Staubli VAL3: _incrementCol.pgx

program _incrementCol(string& x_sColValue[], bool& x_bError[])
  local num l_nColAsciiCode
begin
  x_sColValue=chr((asc(x_sColValue,0)+1))
  call checkColValue(x_sColValue,x_bError)
end
